{attribute addProperty BoxType "EP4378-1022-0017"}
{attribute addProperty Id "Analog_outputAT %Q*INT162"}
{attribute addProperty CRC "4118783225"}
{attribute addProperty SizeInBites "16"}
{attribute addProperty SizeInBytes "2"}
TYPE AO_X06_Pin5_Standard_F57FA4F9 :
STRUCT
	{attribute addProperty Name "Analog_output"}
	Analog_output AT %Q* : INT;
END_STRUCT
END_TYPE

(* stored: Version 1.2.0.0, ProductVersion 3.1.4024.9
   DUT AO_X06_Pin5_Standard_F57FA4F9: Id {cbc80e50-3afe-4b66-b4d6-6d823481ae99} *)
